PROGRAM dbg_lowest
VAR
END_VAR

IF NOT framework_is_local_simulated()
THEN
	RETURN;	
END_IF

END_PROGRAM

(* stored: Version 1.1.0.1, ProductVersion 3.1.4022.12
   POU dbg_lowest: Id {5b454e71-93ca-405f-b31d-bbc38f0ad8e1}, SpecialFunc None *)
